(* Logix 5000 project; controller OptixTest vendor 1 type 14 code 164 rev 37.11; software revision 37.00 *)

TASK MainTask (continuous, watchdog 500 ms) : MainProgram

MODULES
   Local : vendor 1 type 14 code 164 (ICP 2, rev 37.11)
END_MODULES

TYPE Estate :
STRUCT
   Running : BOOL;
   Stop : BOOL;
   Hold : BOOL;
   Alarm : BOOL;
END_STRUCT
END_TYPE

VAR_GLOBAL   (* controller tags *)
   AcumuladordeMoldes : INT;
   Amasadora1 : INT;
   Amasadora2 : INT;
   Apilador : INT;
   Camara_de_Vapor : INT;
   Cortadora : INT;
   Desapilador : INT;
   Desmoldeador : INT;
   Embolsado : INT;
   EmbolsadoraVertical1 : INT;
   EmbolsadoraVertical3 : INT;
   EmbolsadorVertical2 : INT;
   Enfriador : INT;
   HornoBajoCamara : INT;
   Inyectora1 : INT;
   LavadoradeMoldes : INT;
   Receta : BOOL;
   SistemaMOPA : INT;
   Transportador1aCamara : INT;
   Transportador2aCamara : INT := 1;
   TransportadoraEmbolsadoVertical : INT;
   TransportadoraEnvoltura : INT;
   TransportadorAlimentadorMoldes : INT;
   TransportadoraSalidaCortadora : INT;
   TransportadordeDescarga : INT;
   TransportadordeDistribucion : INT;
   TransportadordeSalidaLavadora : INT;
   TransportadoresaApiladores : INT;
   TransportadorInyector : INT;
   TransportadorMoldes : INT;
   TransportadorSalidaHorno : INT;
   TransportadorSalidaMOPA : INT;
   TransportadorTolva : INT;
   TrendeEmbolsado1 : INT;
   TrendeEmbolsado2 : INT;
   TrendeEmbolsado3 : INT;
   TrendeEmbolsado4 : INT;
   TrendeLaminado1 : INT;
   TrendeLaminado2 : INT;
END_VAR

PROGRAM MainProgram   (* main routine MainRoutine *)

ROUTINE MainRoutine   (* ladder *)
END_ROUTINE
END_PROGRAM
